PROGRAM PRG_RecipeList1_1
VAR_INPUT
		bFirst			: BOOL := TRUE;
END_VAR
VAR
	fbEnum				: FB_EnumFindFileList;
	filesList 			: ARRAY[0..99]  OF ST_FindFileEntry;
	bNext				: BOOL;
	bAbort				: BOOL;
	bBusy				: BOOL;
	bError				: BOOL;
	nErrID				: UDINT;
	bEOE				: BOOL;
	nFindFiles			: UDINT;
END_VAR

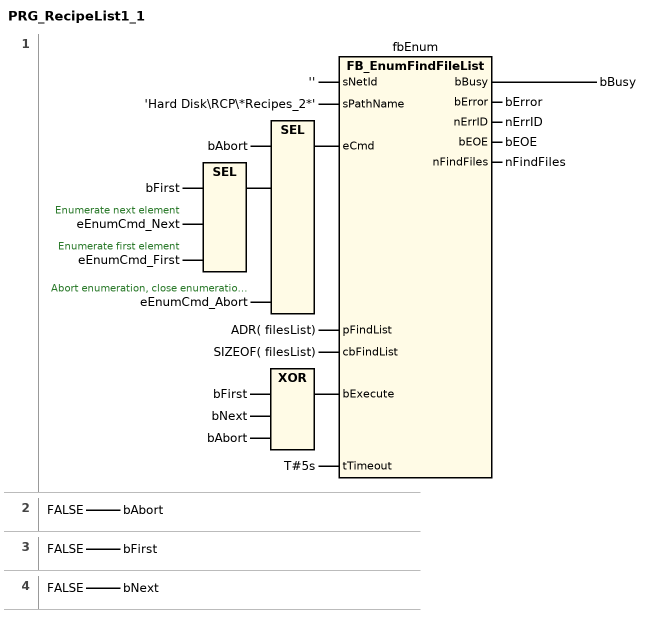
// NETWORK 1
//   eEnumCmd_Next: Enumerate next element
//   eEnumCmd_First: Enumerate first element
//   eEnumCmd_Abort: Abort enumeration, close enumeration handle.
fbEnum(
    sNetId := '',
    sPathName := 'Hard Disk\RCP\*Recipes_2*',
    eCmd := SEL(bAbort, SEL(bFirst, eEnumCmd_Next, eEnumCmd_First), eEnumCmd_Abort),
    pFindList := ADR( filesList),
    cbFindList := SIZEOF( filesList),
    bExecute := bFirst XOR bNext XOR bAbort,
    tTimeout := T#5s,
    bError => bError,
    nErrID => nErrID,
    bEOE => bEOE,
    nFindFiles => nFindFiles); // FB_EnumFindFileList
bBusy := fbEnum.bBusy;

// NETWORK 2
bAbort := FALSE;

// NETWORK 3
bFirst := FALSE;

// NETWORK 4
bNext := FALSE;

END_PROGRAM

(* stored: Version 1.1.0.1, ProductVersion 3.1.4024.12
   POU PRG_RecipeList1_1: Id {232c1344-d262-454c-b219-6011b11177f3}, SpecialFunc None *)
